// TIA Portal project "CP1616_IO_Controller_tutorial_project" (V13)

(* hardware
DEVICE "S7-1200 station_1"  S7-1200 Station
   slot 0: "Rack_0"  Rack  V1.0
   slot 1: "PLC_1"  CPU 1217C DC/DC/DC  6ES7 217-1AG40-0XB0  V4.0
DEVICE "PC-System_1"  SIMATIC PC station
   slot 0: "SIMATIC PC station"  Rail  SIMATIC PC-Station  V1.0
      slot 125: "Stationmanager"  Station_Manager  V6.0.4
   slot 1: "CP 1616_1"  CP 1616  6GK1 161-6AA00  V2.6
*)

// ===== PLC "PLC_1"  CPU 1217C DC/DC/DC =====

VAR_GLOBAL   // PLC tag table "Tag table"
   "CP_input_byte" AT %QB2 : Byte;
   "CP_output_byte" AT %IB2 : Byte;
   "CP_input_real" AT %QD4 : Real;
   "CP_output_real" AT %ID4 : Real;
   "CP_input_byte_array_0" AT %QB8 : Byte;
   "CP_input_byte_array_1" AT %QB9 : Byte;
   "CP_input_byte_array_2" AT %QB10 : Byte;
   "CP_input_byte_array_3" AT %QB11 : Byte;
   "CP_input_byte_array_4" AT %QB12 : Byte;
   "CP_input_byte_array_5" AT %QB13 : Byte;
   "CP_input_byte_array_6" AT %QB14 : Byte;
   "CP_input_byte_array_7" AT %QB15 : Byte;
   "CP_output_byte_array_0" AT %IB8 : Byte;
   "CP_output_byte_array_1" AT %IB9 : Byte;
   "CP_output_byte_array_2" AT %IB10 : Byte;
   "CP_output_byte_array_3" AT %IB11 : Byte;
   "CP_output_byte_array_4" AT %IB12 : Byte;
   "CP_output_byte_array_5" AT %IB13 : Byte;
   "CP_output_byte_array_6" AT %IB14 : Byte;
   "CP_output_byte_array_7" AT %IB15 : Byte;
END_VAR

ORGANIZATION_BLOCK "Main"   // OB1, LAD, ProgramCycle
TITLE = "Main Program Sweep (Cycle)"
{ S7_Optimized_Access := 'FALSE' }
VERSION : 0.1
BEGIN
END_ORGANIZATION_BLOCK